Staubli VAL3: ros_server.pjx

--- ros_server.pjx ---
Parameters version=s8.12Cs9_BS2378 stackSize=5000 millimeterUnit=true
Program file=dataReceiver.pgx
Program file=dataStreamer.pgx
Program file=decodeMsgBody.pgx
Program file=decodeMsgHeader.pgx
Program file=decTrajPt.pgx
Program file=decTrajPtFull.pgx
Program file=encodeAck.pgx
Program file=encodeJState.pgx
Program file=encodeStatus.pgx
Program file=encPrefixHeader.pgx
Program file=encTrajPtAck.pgx
Program file=encTrajPtFAck.pgx
Program file=fetchStatus.pgx
Program file=initParams.pgx
Program file=interpolateVel.pgx
Program file=motionControl.pgx
Program file=pushMotion.pgx
Program file=recvData.pgx
Program file=recvHeartbeat.pgx
Program file=recvMsgBody.pgx
Program file=recvMsgHeader.pgx
Program file=recvTrajPt.pgx
Program file=recvTrajPtFull.pgx
Program file=screenUpdate.pgx
Program file=sendAck.pgx
Program file=sendData.pgx
Program file=sendRosMsg.pgx
Program file=setupRosMsgs.pgx
Program file=start.pgx
Program file=stop.pgx
Program file=taskManager.pgx
Program file=toJointArrayRad.pgx
Program file=toJointRxDeg.pgx
Data file=ros_server.dtx
Library alias=libQueueFuncs path=Disk://ros_libs/QueueFuncs/QueueFuncs.pjx
Library alias=libInterface path=Disk://ros_libs/UserInterface/interfaceDefault/interfaceDefault.pjx autoload=false
Type name=RosSimpleMsg path=Disk://ros_libs/RosSimpleMsg/RosSimpleMsg.pjx
Type name=RobotStatusMsg path=Disk://ros_libs/RobotStatusMsg/RobotStatusMsg.pjx
Type name=JointStateMsg path=Disk://ros_libs/JointStateMsg/JointStateMsg.pjx
Type name=JointTrajPtMsg path=Disk://ros_libs/JointTrajPtMsg/JointTrajPtMsg.pjx
Type name=JointTrajPtFMsg path=Disk://ros_libs/JointTrajPtFMsg/JointTrajPtFMsg.pjx
Type name=JointFbkMsg path=Disk://ros_libs/JointFbkMsg/JointFbkMsg.pjx
Type name=MotionCmd path=Disk://ros_libs/MotionCmd/MotionCmd.pjx
Type name=Header path=Disk://ros_libs/Header/Header.pjx
Type name=Prefix path=Disk://ros_libs/Prefix/Prefix.pjx
Type name=Body path=Disk://ros_libs/Body/Body.pjx
Type name=Queue path=Disk://ros_libs/Queue/Queue.pjx

--- ros_server.dtx ---
public bool bFbkOverrun
public bool bMotionOverrun
public sio siTcpIpFbk = {link=Socket\Feedback}
public sio siTcpIpMotion = {link=Socket\Motion}
public string sStreamTaskName = "publisher"
public string sMotionTaskName
public RosSimpleMsg rosGenericMsg
  [0]
    Header header
      [0]
        num nMsgType
        num nCommType
        num nReplyCode
        num nData[12]
    Prefix prefix
      [0]
        num nLength
        num nData[4]
public tool tTool = {fatherId=flange[0], ioLink=ValveIO\valve1}
public string sTrajPtTaskName
public bool bTrajPtOverrun
public RobotStatusMsg rosStatusMsg
  [0]
    Body body
      [0]
        num nData[28]
    Header header
      [0]
        num nMsgType
        num nCommType
        num nReplyCode
        num nData[12]
    Prefix prefix
      [0]
        num nLength
        num nData[4]
    RobotStatus robotStatus
      [0]
        num nDrivesPowered
        num nEStopped
        num nErrorCode
        num nInError
        num nInMotion
        num nMode
        num nMotionPossible
public JointStateMsg rosJointMsg
  [0]
    Header header
      [0]
        num nMsgType
        num nCommType
        num nReplyCode
        num nData[12]
    Body body
      [0]
        num nData[44]
    JointState jointState
      [0]
        num nSeq
        num nJoints[10]
    Prefix prefix
      [0]
        num nLength
        num nData[4]
public JointTrajPtMsg rosTrajPtMsg
  [0]
    Header header
      [0]
        num nMsgType
        num nCommType
        num nReplyCode
        num nData[12]
    JointTrajPt jointTrajPt
      [0]
        num nSeq
        num nJoints[10]
        num nVelocity
        num nDuration
    Prefix prefix
      [0]
        num nLength
        num nData[4]
    Body body
      [0]
        num nData[52]
public JointTrajPtFMsg rosTrajPtFMsg
  [0]
    Header header
      [0]
        num nMsgType
        num nCommType
        num nReplyCode
        num nData[12]
    Prefix prefix
      [0]
        num nLength
        num nData[4]
    JointTrajPtFull jointTrajPtFull
      [0]
        num nRobotId
        num nSeq
        num nValidFields
        num nTime
        num nPositions[10]
        num nVelocities[10]
        num nAccelerations[10]
    Body body
      [0]
        num nData[136]
public JointFbkMsg rosJointFbkMsg
  [0]
    Header header
      [0]
        num nMsgType
        num nCommType
        num nReplyCode
        num nData[12]
    Prefix prefix
      [0]
        num nLength
        num nData[4]
    JointFeedback jointFeedback
      [0]
        num nRobotId
        num nValidFields
        num nTime
        num nPositions[10]
        num nVelocities[10]
        num nAccelerations[10]
    Body body
      [0]
        num nData[132]
public JointTrajPtFMsg rosTrajPtFAck
  [0]
    Header header
      [0]
        num nMsgType
        num nCommType
        num nReplyCode
        num nData[12]
    Prefix prefix
      [0]
        num nLength
        num nData[4]
    JointTrajPtFull jointTrajPtFull
      [0]
        num nRobotId
        num nSeq
        num nValidFields
        num nTime
        num nPositions[10]
        num nVelocities[10]
        num nAccelerations[10]
    Body body
      [0]
        num nData[136]
public JointTrajPtMsg rosTrajPtAck
  [0]
    Header header
      [0]
        num nMsgType
        num nCommType
        num nReplyCode
        num nData[12]
    JointTrajPt jointTrajPt
      [0]
        num nSeq
        num nJoints[10]
        num nVelocity
        num nDuration
    Prefix prefix
      [0]
        num nLength
        num nData[4]
    Body body
      [0]
        num nData[52]
public bool bScreenOverrun
public string sScreenTaskName
public num nInConnFlag
public num nOutConnFlag
public string sHtbtTaskName
public num nPtsPopped
public bool bStopNow
public num nMotionProgress
public num nMoveId
public num nMovePts
public num nElapsedTime
public num nHeaderTime
public bool bOverwriteVel
public Queue qMoveBuffer
  [0]
    num nPush
    num nPop
    num nElems
    MotionCmd buffer[10]
      [0]
        mdesc mDesc = {leave=0, reach=0}
        num nDuration
        num nSequence
        jointRx jJointRx
      [1]
        mdesc mDesc = {leave=0, reach=0}
        num nDuration
        num nSequence
        jointRx jJointRx
      [2]
        mdesc mDesc = {leave=0, reach=0}
        num nDuration
        num nSequence
        jointRx jJointRx
      [3]
        mdesc mDesc = {leave=0, reach=0}
        num nDuration
        num nSequence
        jointRx jJointRx
      [4]
        mdesc mDesc = {leave=0, reach=0}
        num nDuration
        num nSequence
        jointRx jJointRx
      [5]
        mdesc mDesc = {leave=0, reach=0}
        num nDuration
        num nSequence
        jointRx jJointRx
      [6]
        mdesc mDesc = {leave=0, reach=0}
        num nDuration
        num nSequence
        jointRx jJointRx
      [7]
        mdesc mDesc = {leave=0, reach=0}
        num nDuration
        num nSequence
        jointRx jJointRx
      [8]
        mdesc mDesc = {leave=0, reach=0}
        num nDuration
        num nSequence
        jointRx jJointRx
      [9]
        mdesc mDesc = {leave=0, reach=0}
        num nDuration
        num nSequence
        jointRx jJointRx
public Queue qTrajPtBuffer
  [0]
    num nPush
    num nPop
    num nElems
    MotionCmd buffer[10]
      [0]
        mdesc mDesc = {leave=0, reach=0}
        num nDuration
        num nSequence
        jointRx jJointRx
      [1]
        mdesc mDesc = {leave=0, reach=0}
        num nDuration
        num nSequence
        jointRx jJointRx
      [2]
        mdesc mDesc = {leave=0, reach=0}
        num nDuration
        num nSequence
        jointRx jJointRx
      [3]
        mdesc mDesc = {leave=0, reach=0}
        num nDuration
        num nSequence
        jointRx jJointRx
      [4]
        mdesc mDesc = {leave=0, reach=0}
        num nDuration
        num nSequence
        jointRx jJointRx
      [5]
        mdesc mDesc = {leave=0, reach=0}
        num nDuration
        num nSequence
        jointRx jJointRx
      [6]
        mdesc mDesc = {leave=0, reach=0}
        num nDuration
        num nSequence
        jointRx jJointRx
      [7]
        mdesc mDesc = {leave=0, reach=0}
        num nDuration
        num nSequence
        jointRx jJointRx
      [8]
        mdesc mDesc = {leave=0, reach=0}
        num nDuration
        num nSequence
        jointRx jJointRx
      [9]
        mdesc mDesc = {leave=0, reach=0}
        num nDuration
        num nSequence
        jointRx jJointRx
num nVel[2]
num nStdMsgType{}
  [JOINT_TRAJ_PT] = 11
  [JOINT_TRAJ_PT_FULL] = 14
num nCommType{}
  [SERVICE_REQUEST] = 2
mdesc mNomSpeed
num nRecHeader
num nDecHeader = 1
num nRecBody = 2
num nDecBody = 3
num nPushMotion = 4
num nAck = 5
num nReset
num nFbkPeriod
num nMotionPeriod
num nTrajPeriod
num nScreenUpdate
num nFbkOverun
num nTrajPtOverrun
num nMotionOverrun
num nLibLoadError

--- start.pgx ---
program start()
  local num l_nScreenUpdate
  local string l_sVersionMajor
  local num l_nVersionMajor
  local bool l_bOkMajor
  local string l_sVersionMinor
  local num l_nVersionMinor
  local bool l_bOkMinor
  local num l_nLibLoad
begin
  // Copyright (c) 2016, Ocado Technology - Robotics Research Team
  //
  // Licensed under the Apache License, Version 2.0 (the "License");
  // you may not use this file except in compliance with the License.
  // You may obtain a copy of the License at
  //
  //     http://www.apache.org/licenses/LICENSE-2.0
  //
  // Unless required by applicable law or agreed to in writing, software
  // distributed under the License is distributed on an "AS IS" BASIS,
  // WITHOUT WARRANTIES OR CONDITIONS OF ANY KIND, either express or implied.
  // See the License for the specific language governing permissions and
  // limitations under the License.


  // Load interface library for CS8 or CS9
  //
  // CS9 handles the UI differently than CS8, requires
  // the UI funtions to be loaded in seperate libraries

  if(mid(getVersion("System"),1,1) == "7")
    // CS8 - VAL 3 rev 7
    // Check for VAL 3 version >= 7.7
    l_sVersionMajor = mid(getVersion("VAL3"),1,1)
    l_sVersionMinor = mid(getVersion("VAL3"),2,1)
    toNum(l_sVersionMajor, l_nVersionMajor, l_bOkMajor)
    toNum(l_sVersionMinor, l_nVersionMinor, l_bOkMinor)
    if(!l_bOkMajor or !l_bOkMinor)
      popUpMsg("Error reading VAL 3 version")
      call stop()
    endIf
    if( !((l_nVersionMajor == 7) and (l_nVersionMinor >= 7)))
      // VAL 3 version is too old
      popUpMsg("Error: VAL 3 version is < 7.7, socket communication will not work!")
      call stop()
    endIf
    nLibLoadError = libInterface:libLoad("ros_libs/UserInterface/interfaceCS8")
  elseIf(mid(getVersion("System"),1,1) == "8")
    // CS9 - VAL 3 rev 8
    nLibLoadError = libInterface:libLoad("ros_libs/UserInterface/interfaceCS9")
  endIf

  // check for libLoad error
  if nLibLoadError != 0
    popUpMsg("Error loading UserPage!")
    call stop()
  else
    // feedback task will run every 20ms (50Hz)
    nFbkPeriod=0.02
    //l_nFbkPeriod = 0.032 // 30Hz
    //l_nFbkPeriod = 0.05  // 20Hz
    //l_nFbkPeriod = 1.0   //  1Hz

    // motion control task will run every 4ms (250Hz)
    nMotionPeriod = 0.004
    //l_nMotionPeriod=0.012  // 83Hz
    //l_nMotionPeriod = 0.05 // 20Hz

    // data (trajectory) reception task will run every 4ms (250Hz)
    nTrajPeriod = 0.004
    // not in use at the moment
    nScreenUpdate = 1.0

    sStreamTaskName = "streamerTask"
    sTrajPtTaskName = "trajPtTask"
    sMotionTaskName = "motionTask"
    sScreenTaskName = "screenTask"
    sHtbtTaskName = "htbtTask"

    // initialise TCP/IP parameters
    call initParams()
    // setup prefix and header of ROS messages
    call setupRosMsgs()

    // socket connection status flags: initially disconnected
    nInConnFlag = 0
    nOutConnFlag = 0

    // flag defining whether velocity to be overwritten to max. vel.
    bOverwriteVel = false

    nPtsPopped = 0
    nMovePts = 0

    // flush buffer of incoming socket
    clearBuffer(siTcpIpMotion)
    // flush buffer of outgoing socket
    clearBuffer(siTcpIpFbk)

    // check if robot is not in emergency stop and wait until estop is reset
    if(esStatus() == 2)
      popUpMsg("Please reset E-Stop")
      wait(esStatus() < 2)
    endIf

    // before anything else, enable power (only works if robot is in remote mode)
    if(!isPowered())
      if(workingMode() >= 4)
        do
          enablePower()
          delay(2)
        until isPowered()
      else
        popUpMsg("Power must be enabled manually")
      endIf
    endIf

    // reset motion, potentially setting a start joint position for calling autoConnect() in the future
    resetMotion()

    //start task for the taskManager:
    taskCreate "taskManager", 50, taskManager()
    wait(taskStatus("taskManager") != -1)
  endIf


end

--- dataReceiver.pgx ---
public program dataReceiver()
  local num l_nStartTime
  local num l_nMsgRecvState
begin
  // Copyright (c) 2016, Ocado Technology - Robotics Research Team
  //
  // Licensed under the Apache License, Version 2.0 (the "License");
  // you may not use this file except in compliance with the License.
  // You may obtain a copy of the License at
  //
  //     http://www.apache.org/licenses/LICENSE-2.0
  //
  // Unless required by applicable law or agreed to in writing, software
  // distributed under the License is distributed on an "AS IS" BASIS,
  // WITHOUT WARRANTIES OR CONDITIONS OF ANY KIND, either express or implied.
  // See the License for the specific language governing permissions and
  // limitations under the License.



  // state machine at initial state
  // 0: receive header
  // 1: decode header
  // 2: receive body
  // 3: decode body
  // 4: push motion into buffer
  // 5: send ACK

  // Set variable constants to make sure they were not changed
  nReset=0
  nRecHeader=0
  nDecHeader=1
  nRecBody=2
  nDecBody=3
  nPushMotion=4
  nAck=5

  l_nMsgRecvState=nRecHeader

  while(true)
    // usually for state machines a switch-case statement is a neat implementation
    // HOWEVER, at every iteration of while() this task is sequenced and only called
    // after whatever ms is was defined when created.
    // As a result, receiving one single message, pushing motion and sending ACK
    // would take 6 * task period using switch-case statement.
    // The desirable behaviour is to receive and decode a full message, push motion
    // into buffer and then send ACK to client WITHIN ONE ITERATION of while(),
    // hence the if statement sequence below

        // check for overrun
    if bTrajPtOverrun
      nTrajPtOverrun = nTrajPtOverrun + 1
    endIf


    l_nStartTime = clock()
    if(l_nMsgRecvState==nRecHeader)
      call recvMsgHeader(l_nMsgRecvState)
    endIf
    nHeaderTime = clock() - l_nStartTime
    if(l_nMsgRecvState==nDecHeader)
      call decodeMsgHeader(l_nMsgRecvState)
    endIf
    if(l_nMsgRecvState==nRecBody)
      call recvMsgBody(l_nMsgRecvState)
    endIf
    if(l_nMsgRecvState==nDecBody)
      call decodeMsgBody(l_nMsgRecvState)
    endIf
    if(l_nMsgRecvState==nPushMotion)
      call pushMotion(l_nMsgRecvState)
    endIf
    if(l_nMsgRecvState==nAck)
      call encodeAck()
      call sendAck(l_nMsgRecvState)
    endIf
    nElapsedTime = clock() - l_nStartTime - nHeaderTime

    // assert state machine is working OK
    if(l_nMsgRecvState<nRecHeader or l_nMsgRecvState>nAck)
      popUpMsg("Data reception state machine error")
    endIf

    // sequence task
    delay(0)


  endWhile
end

--- dataStreamer.pgx ---
public program dataStreamer()
  local num l_nThrottle
  local jointRx l_jCurrPose
begin
  // Copyright (c) 2016, Ocado Technology - Robotics Research Team
  //
  // Licensed under the Apache License, Version 2.0 (the "License");
  // you may not use this file except in compliance with the License.
  // You may obtain a copy of the License at
  //
  //     http://www.apache.org/licenses/LICENSE-2.0
  //
  // Unless required by applicable law or agreed to in writing, software
  // distributed under the License is distributed on an "AS IS" BASIS,
  // WITHOUT WARRANTIES OR CONDITIONS OF ANY KIND, either express or implied.
  // See the License for the specific language governing permissions and
  // limitations under the License.



  l_nThrottle = 0
  while(true)
    // check for overrun
    if bFbkOverrun
      nFbkOverun = nFbkOverun + 1
    endIf

    // only attempt to send data if flag indicates that connection is established
      if(nOutConnFlag == 1)
        // fetch current joint positions
        l_jCurrPose=herej()
        // encode and send ROS simple_message ID 10: joint state
        call encodeJState(l_jCurrPose)
        call sendRosMsg(siTcpIpFbk, rosJointMsg.prefix, rosJointMsg.header, rosJointMsg.body, nOutConnFlag)

        // send Robot Status messages 5 times slower than Joint State
        if(l_nThrottle == 5)
          // fetch robot status
          call fetchStatus()
          // encode and send ROS simple_message ID 13: robot status
          call encodeStatus()
          call sendRosMsg(siTcpIpFbk, rosStatusMsg.prefix, rosStatusMsg.header, rosStatusMsg.body, nOutConnFlag)
          l_nThrottle = 0
        endIf
        l_nThrottle = l_nThrottle + 1
      else
        delay(0.1)
      endIf

      // sequence task
      delay(0)
  endWhile
end

--- decodeMsgBody.pgx ---
public program decodeMsgBody(RosSimpleMsg& x_msg, num& x_nMsgRecvState)
  local bool l_bFlag
begin
  // Copyright (c) 2016, Ocado Technology - Robotics Research Team
  // Copyright (c) 2021, Institute for Factory Automation and Production Systems (FAPS)
  //
  // Licensed under the Apache License, Version 2.0 (the "License");
  // you may not use this file except in compliance with the License.
  // You may obtain a copy of the License at
  //
  //     http://www.apache.org/licenses/LICENSE-2.0
  //
  // Unless required by applicable law or agreed to in writing, software
  // distributed under the License is distributed on an "AS IS" BASIS,
  // WITHOUT WARRANTIES OR CONDITIONS OF ANY KIND, either express or implied.
  // See the License for the specific language governing permissions and
  // limitations under the License.


  // assume failure to decode
  l_bFlag=false

  //region @decode -- call specific decode function
  switch x_msg.header.nMsgType
    case SimpleMsg:MsgType.JOINT_TRAJ_PT
      call decTrajPt(l_bFlag)
    break
    case SimpleMsg:MsgType.JOINT_TRAJ_PT_F
      call decTrajPtFull(l_bFlag)
    break
    // Staubli specific
    case Staubli:MsgType.SET_DRIVE_POWER
      call Staubli:decSetDrvPwrMsg(l_bFlag)
    break
    case Staubli:MsgType.WRITE_SINGLE_IO
      call Staubli:decWriSingIOMsg(l_bFlag)
    break
    case Staubli:MsgType.VELOCITY_CFG
      call Staubli:decodeVelCfg(l_bFlag)
    break
    case Staubli:MsgType.VELOCITY_CMD
      call Staubli:decodeVelCmd(l_bFlag)
    break
    default
      //region @DEBUG
      if (bDebugMode and nDebugLevel<=3)
        call printDebug("ERROR: unknown msg type ("+toString("",x_msg.header.nMsgType)+")",false)
        call printDebug("       could not decode message",false)
      endIf
      //endregion
    break
  endSwitch
  //endregion

  //region @check_success -- check whether decoding was successful and move on to the next state
  if (l_bFlag == true)
    switch x_msg.header.nMsgType
      case SimpleMsg:MsgType.JOINT_TRAJ_PT,SimpleMsg:MsgType.JOINT_TRAJ_PT_F,Staubli:MsgType.VELOCITY_CFG,Staubli:MsgType.VELOCITY_CMD
        // move on to state: push motion into buffer
        x_nMsgRecvState = MsgRecvState.PUSH_MOTION
      break
      case Staubli:MsgType.SET_DRIVE_POWER, Staubli:MsgType.WRITE_SINGLE_IO
        // move on to state: handle system/io request
        x_nMsgRecvState = MsgRecvState.HANDLE_REQUEST
      break
    endSwitch

    //region @DEBUG
    if (bDebugMode and nDebugLevel<=3)
      call printDebug("INFO: decoding successful",false)
    endIf
    //endregion
  else
    // error whilst decoding msg body...
    if (x_msg.header.nCommType==SimpleMsg:CommType.SERVICE_REQUEST)
      // set reply code if comm type is request
      switch x_msg.header.nMsgType
        case SimpleMsg:MsgType.JOINT_TRAJ_PT
          rosTrajPtAck.header.nReplyCode=SimpleMsg:ReplyCode.FAILURE
        break
        case SimpleMsg:MsgType.JOINT_TRAJ_PT_F
          rosTrajPtFAck.header.nReplyCode=SimpleMsg:ReplyCode.FAILURE
        break
        // Staubli specific
        case Staubli:MsgType.SET_DRIVE_POWER
          Staubli:setDrvPwrAck.header.nReplyCode=SimpleMsg:ReplyCode.FAILURE
        break
        case Staubli:MsgType.WRITE_SINGLE_IO
          Staubli:writeSingIOAck.header.nReplyCode=SimpleMsg:ReplyCode.FAILURE
        break
        case Staubli:MsgType.VELOCITY_CFG
          Staubli:velCfgAck.header.nReplyCode=SimpleMsg:ReplyCode.FAILURE
        break
        case Staubli:MsgType.VELOCITY_CMD
          Staubli:velCmdAck.header.nReplyCode=SimpleMsg:ReplyCode.FAILURE
        break
        default
          //region @DEBUG
          if (bDebugMode and nDebugLevel<=3)
            call printDebug("ERROR: unknown msg type ("+toString("",x_msg.header.nMsgType)+")",false)
            call printDebug("       could not set reply code",false)
          endIf
          //endregion
        break
      endSwitch
      // jump to state 6: sendAck()
      x_nMsgRecvState = MsgRecvState.SEND_ACK
    else
      // reset state machine, since no ACK is required
      x_nMsgRecvState = MsgRecvState.RECEIVE_HEADER
    endIf
    //region @DEBUG
    if (bDebugMode and nDebugLevel<=3)
      call printDebug("ERROR: decoding not successful",false)
    endIf
    //endregion
  endIf
  //endregion
end

--- decodeMsgHeader.pgx ---
public program decodeMsgHeader(RosSimpleMsg& x_msg (dimensions=1), num& x_nMsgRecvState (dimensions=1))
  local num l_nRetVal
begin
  // Copyright (c) 2016, Ocado Technology - Robotics Research Team
  // Copyright (c) 2021, Institute for Factory Automation and Production Systems (FAPS)
  //
  // Licensed under the Apache License, Version 2.0 (the "License");
  // you may not use this file except in compliance with the License.
  // You may obtain a copy of the License at
  //
  //     http://www.apache.org/licenses/LICENSE-2.0
  //
  // Unless required by applicable law or agreed to in writing, software
  // distributed under the License is distributed on an "AS IS" BASIS,
  // WITHOUT WARRANTIES OR CONDITIONS OF ANY KIND, either express or implied.
  // See the License for the specific language governing permissions and
  // limitations under the License.



  // decode message into generic message first
  l_nRetVal=fromBinary(x_msg.prefix.nData,4,"-4l",x_msg.prefix.nLength)
  if (l_nRetVal!=1)
    // error decoding prefix, reset state machine
    x_nMsgRecvState = MsgRecvState.RECEIVE_HEADER
    return
  endIf
  l_nRetVal=fromBinary(x_msg.header.nData,4,"-4l",x_msg.header.nMsgType)
  if (l_nRetVal!=1)
    // error decoding header (msg type), reset state machine
    x_nMsgRecvState = MsgRecvState.RECEIVE_HEADER
    return
  endIf
  l_nRetVal=fromBinary(x_msg.header.nData[4],4,"-4l",x_msg.header.nCommType)
  if (l_nRetVal!=1)
    // error decoding header (comm type), reset state machine
    x_nMsgRecvState = MsgRecvState.RECEIVE_HEADER
    return
  endIf
  l_nRetVal=fromBinary(x_msg.header.nData[8],4,"-4l",x_msg.header.nReplyCode)
  if (l_nRetVal!=1)
    // error decoding header (reply code), reset state machine
    x_nMsgRecvState = MsgRecvState.RECEIVE_HEADER
    return
  endIf

  // no errors detected whilst decoding prefix and header
  // move on to state 2: receive msg body
  x_nMsgRecvState = MsgRecvState.RECEIVE_BODY

  // debug
  if (bDebugMode and nDebugLevel<=1)
    call printDebug("decodeMsgHeader: successful",true)
    call printDebug("Prefix    :"+toString("",x_msg.prefix.nLength),false)
    call printDebug("MsgType   :"+toString("",x_msg.header.nMsgType),false)
    call printDebug("CommType  :"+toString("",x_msg.header.nCommType),false)
    call printDebug("ReplyType :"+toString("",x_msg.header.nReplyCode),false)
  endIf
end

--- decTrajPt.pgx ---
public program decTrajPt(bool& x_bFlag)
  local num l_nIndex
  local num l_nRetVal
begin
  // Copyright (c) 2016, Ocado Technology - Robotics Research Team
  //
  // Licensed under the Apache License, Version 2.0 (the "License");
  // you may not use this file except in compliance with the License.
  // You may obtain a copy of the License at
  //
  //     http://www.apache.org/licenses/LICENSE-2.0
  //
  // Unless required by applicable law or agreed to in writing, software
  // distributed under the License is distributed on an "AS IS" BASIS,
  // WITHOUT WARRANTIES OR CONDITIONS OF ANY KIND, either express or implied.
  // See the License for the specific language governing permissions and
  // limitations under the License.



  // decode message ID 11 body (data)

  // assume failure to decode
  rosTrajPtAck.header.nReplyCode=2

  // sequence
  l_nRetVal=fromBinary(rosTrajPtMsg.body.nData,4,"-4l",rosTrajPtMsg.jointTrajPt.nSeq)
  if(l_nRetVal!=1)
    x_bFlag=false
    return
  endIf

  // joints[10]
  for l_nIndex=0 to 9 step 1
    l_nRetVal=fromBinary(rosTrajPtMsg.body.nData[(l_nIndex*4)+4],4,"4.0l",rosTrajPtMsg.jointTrajPt.nJoints[l_nIndex])
    if(l_nRetVal!=1)
      x_bFlag=false
      return
    endIf
  endFor

  // velocity
  l_nRetVal=fromBinary(rosTrajPtMsg.body.nData[44],4,"4.0l",rosTrajPtMsg.jointTrajPt.nVelocity)
  if(l_nRetVal!=1)
    x_bFlag=false
    return
  endIf

  // duration
  l_nRetVal=fromBinary(rosTrajPtMsg.body.nData[48],4,"4.0l",rosTrajPtMsg.jointTrajPt.nDuration)
  if(l_nRetVal!=1)
    x_bFlag=false
    return
  endIf

  // decoding successful
  rosTrajPtAck.header.nReplyCode=1
  rosTrajPtAck.jointTrajPt.nSeq=rosTrajPtMsg.jointTrajPt.nSeq
  x_bFlag=true
end

--- decTrajPtFull.pgx ---
public program decTrajPtFull(bool& x_bFlag)
  local num l_nIndex
  local num l_nRetVal
begin
  // Copyright (c) 2016, Ocado Technology - Robotics Research Team
  //
  // Licensed under the Apache License, Version 2.0 (the "License");
  // you may not use this file except in compliance with the License.
  // You may obtain a copy of the License at
  //
  //     http://www.apache.org/licenses/LICENSE-2.0
  //
  // Unless required by applicable law or agreed to in writing, software
  // distributed under the License is distributed on an "AS IS" BASIS,
  // WITHOUT WARRANTIES OR CONDITIONS OF ANY KIND, either express or implied.
  // See the License for the specific language governing permissions and
  // limitations under the License.



  // decode message ID 14 body (data)

  // assume failure to decode
  rosTrajPtFAck.header.nReplyCode=2

  // robotId
  l_nRetVal=fromBinary(rosTrajPtFMsg.body.nData,4,"-4l",rosTrajPtFMsg.jointTrajPtFull.nRobotId)
  if(l_nRetVal!=1)
    x_bFlag=false
    return
  endIf

  // sequence
  l_nRetVal=fromBinary(rosTrajPtFMsg.body.nData,4,"-4l",rosTrajPtFMsg.jointTrajPtFull.nSeq)
  if(l_nRetVal!=1)
    x_bFlag=false
    return
  endIf

  // valid fields
  l_nRetVal=fromBinary(rosTrajPtFMsg.body.nData,4,"-4l",rosTrajPtFMsg.jointTrajPtFull.nValidFields)
  if(l_nRetVal!=1)
    x_bFlag=false
    return
  endIf

  // time
  l_nRetVal=fromBinary(rosTrajPtFMsg.body.nData,4,"4.0l",rosTrajPtFMsg.jointTrajPtFull.nTime)
  if(l_nRetVal!=1)
    x_bFlag=false
    return
  endIf

  // positions[10]
  for l_nIndex=0 to 9 step 1
    l_nRetVal=fromBinary(rosTrajPtFMsg.body.nData[(l_nIndex*4)+16],4,"4.0l",rosTrajPtFMsg.jointTrajPtFull.nPositions[l_nIndex])
    if(l_nRetVal!=1)
      x_bFlag=false
      return
    endIf
  endFor

  // velocities[10]
  for l_nIndex=0 to 9 step 1
    l_nRetVal=fromBinary(rosTrajPtFMsg.body.nData[(l_nIndex*4)+56],4,"4.0l",rosTrajPtFMsg.jointTrajPtFull.nVelocities[l_nIndex])
    if(l_nRetVal!=1)
      x_bFlag=false
      return
    endIf
  endFor

  // accelerations[10]
  for l_nIndex=0 to 9 step 1
    l_nRetVal=fromBinary(rosTrajPtFMsg.body.nData[(l_nIndex*4)+96],4,"4.0l",rosTrajPtFMsg.jointTrajPtFull.nAccelerations[l_nIndex])
    if(l_nRetVal!=1)
      x_bFlag=false
      return
    endIf
  endFor

  // decoding successful
  rosTrajPtFAck.header.nReplyCode=1
  rosTrajPtFAck.jointTrajPtFull.nSeq=rosTrajPtFMsg.jointTrajPtFull.nSeq
  x_bFlag=true
end

--- encodeAck.pgx ---
public program encodeAck(RosSimpleMsg& x_msg)
begin
  // Copyright (c) 2016, Ocado Technology - Robotics Research Team
  // Copyright (c) 2021, Institute for Factory Automation and Production Systems (FAPS)
  //
  // Licensed under the Apache License, Version 2.0 (the "License");
  // you may not use this file except in compliance with the License.
  // You may obtain a copy of the License at
  //
  //     http://www.apache.org/licenses/LICENSE-2.0
  //
  // Unless required by applicable law or agreed to in writing, software
  // distributed under the License is distributed on an "AS IS" BASIS,
  // WITHOUT WARRANTIES OR CONDITIONS OF ANY KIND, either express or implied.
  // See the License for the specific language governing permissions and
  // limitations under the License.



  switch x_msg.header.nMsgType

    case SimpleMsg:MsgType.JOINT_TRAJ_PT
      call encTrajPtAck()
    break

    case SimpleMsg:MsgType.JOINT_TRAJ_PT_F
      call encTrajPtFAck()
    break

    // Staubli specific
    case Staubli:MsgType.SET_DRIVE_POWER
      call Staubli:encSetDrvPwrAck()
    break

    case Staubli:MsgType.WRITE_SINGLE_IO
      call Staubli:encWriSingIOAck()
    break

    case Staubli:MsgType.VELOCITY_CFG
      call Staubli:encodeVelCfgAck()
    break

    case Staubli:MsgType.VELOCITY_CMD
      call Staubli:encodeVelCmdAck()
    break

    default
      //region @DEBUG
      if (bDebugMode and nDebugLevel<=5)
        call printDebug("encodeAck: switch (msgType)",true)
        call printDebug("ERROR: unknown msg type",false)
      endIf
      //endregion
    break
  endSwitch
end

--- encodeJFeedback.pgx ---
program encodeJFeedback(num x_nTime, jointRx x_jPosition, jointRx x_jVelocity)
begin
  // Copyright (c) 2021, Institute for Factory Automation and Production Systems (FAPS)
  //
  // Licensed under the Apache License, Version 2.0 (the "License");
  // you may not use this file except in compliance with the License.
  // You may obtain a copy of the License at
  //
  //     http://www.apache.org/licenses/LICENSE-2.0
  //
  // Unless required by applicable law or agreed to in writing, software
  // distributed under the License is distributed on an "AS IS" BASIS,
  // WITHOUT WARRANTIES OR CONDITIONS OF ANY KIND, either express or implied.
  // See the License for the specific language governing permissions and
  // limitations under the License.


  // encode 'prefix' and 'header'
  call encPrefixHeader(rosJointFbkMsg.prefix, rosJointFbkMsg.header)

  // encode 'robot_id' variable of body message (data)
  toBinary(rosJointFbkMsg.jointFeedback.nRobotId, 1, "-4l", rosJointFbkMsg.body.nData)

  // encode 'valid_fields' variable of body message (data)
  toBinary(rosJointFbkMsg.jointFeedback.nValidFields, 1, "-4l", rosJointFbkMsg.body.nData[4])

  // encode 'time' variable of body message (data)
  toBinary(rosJointFbkMsg.jointFeedback.nTime, 1, "-4l", rosJointFbkMsg.body.nData[8])

  call toJointArrayRad(x_jPosition, rosJointFbkMsg.jointFeedback.nPositions)

  // encode 10 values representing joint positions [10]
  toBinary(rosJointFbkMsg.jointFeedback.nPositions, 10, "4.0l", rosJointFbkMsg.body.nData[12])

  call toJointArrayRad(x_jVelocity, rosJointFbkMsg.jointFeedback.nVelocities)

  // encode 10 values representing joint velocities [10]
  toBinary(rosJointFbkMsg.jointFeedback.nVelocities, 10, "4.0l", rosJointFbkMsg.body.nData[52])
end

--- fetchStatus.pgx ---
public program fetchStatus()
begin
  // Copyright (c) 2016, Ocado Technology - Robotics Research Team
  // Copyright (c) 2021, Institute for Factory Automation and Production Systems (FAPS)
  //
  // Licensed under the Apache License, Version 2.0 (the "License");
  // you may not use this file except in compliance with the License.
  // You may obtain a copy of the License at
  //
  //     http://www.apache.org/licenses/LICENSE-2.0
  //
  // Unless required by applicable law or agreed to in writing, software
  // distributed under the License is distributed on an "AS IS" BASIS,
  // WITHOUT WARRANTIES OR CONDITIONS OF ANY KIND, either express or implied.
  // See the License for the specific language governing permissions and
  // limitations under the License.



  // fetch robot status data

  // drives_powered
  if (isPowered()==true)
    rosStatusMsg.robotStatus.nDrivesPowered=1
  else
    rosStatusMsg.robotStatus.nDrivesPowered=0
  endIf

  // e-stopped
  if (esStatus()==2)
    rosStatusMsg.robotStatus.nEStopped=1
  else
    rosStatusMsg.robotStatus.nEStopped=0
  endIf

  // error_code
  if (taskStatus(sMotionTask) > 1)
    rosStatusMsg.robotStatus.nErrorCode = taskStatus(sMotionTask)
  elseIf (taskStatus(sMotionRecvTask) > 1)
    rosStatusMsg.robotStatus.nErrorCode = taskStatus(sMotionRecvTask)
  elseIf (taskStatus(sStreamerTask) > 1)
    rosStatusMsg.robotStatus.nErrorCode = taskStatus(sStreamerTask)
  elseIf (taskStatus(sHeartbeatTask) > 1)
    rosStatusMsg.robotStatus.nErrorCode = taskStatus(sHeartbeatTask)
  elseIf (taskStatus(sScreenTask) > 1)
    rosStatusMsg.robotStatus.nErrorCode = taskStatus(sScreenTask)
  else
    rosStatusMsg.robotStatus.nErrorCode = 0
  endIf

  // in_error
  if (taskStatus(sMotionRecvTask) == 1 and taskStatus(sMotionTask) == 1 and taskStatus(sStreamerTask) == 1 and taskStatus(sScreenTask) == 1 and taskStatus(sHeartbeatTask) == 1)
    rosStatusMsg.robotStatus.nInError = 0
  else
    rosStatusMsg.robotStatus.nInError = 1
  endIf

  // in_motion
  if (isSettled()==true)
    rosStatusMsg.robotStatus.nInMotion=0
  else
    rosStatusMsg.robotStatus.nInMotion=1
  endIf

  // mode (controller/pendant mode)
  // according to industrial_msgs/RobotMode, possible values are:
  // -1: unknown or unavailable
  //  1: teach or manual mode
  //  2: automatic mode (which I interpret as either local or remote)
  if (workingMode() == 0)
    rosStatusMsg.robotStatus.nMode = -1
  elseIf (workingMode()==1 or workingMode()==2)
    rosStatusMsg.robotStatus.nMode = 1
  elseIf (workingMode()==3 or workingMode()==4)
    rosStatusMsg.robotStatus.nMode = 2
  endIf

  // motion_possible:
  // drives must be powered and e-stop must be off
  // and dataReceiver and motionControl tasks must be
  // running normally
  if (isPowered() == true and esStatus() == 0 and taskStatus(sMotionRecvTask) == 1 and taskStatus(sMotionTask) == 1)
    rosStatusMsg.robotStatus.nMotionPossible=1
  else
    rosStatusMsg.robotStatus.nMotionPossible=0
  endIf
end

--- handleRequest.pgx ---
public program handleRequest(RosSimpleMsg& x_msg, num& x_nMsgRecvState)
  local bool l_bOk
  local num l_nModuleId
  local num l_nPin
  local bool l_bState
begin
  // Copyright (c) 2021, Institute for Factory Automation and Production Systems (FAPS)
  //
  // Licensed under the Apache License, Version 2.0 (the "License");
  // you may not use this file except in compliance with the License.
  // You may obtain a copy of the License at
  //
  //     http://www.apache.org/licenses/LICENSE-2.0
  //
  // Unless required by applicable law or agreed to in writing, software
  // distributed under the License is distributed on an "AS IS" BASIS,
  // WITHOUT WARRANTIES OR CONDITIONS OF ANY KIND, either express or implied.
  // See the License for the specific language governing permissions and
  // limitations under the License.


  // assume success to push motion
  l_bOk=true

  // handle request
  switch x_msg.header.nMsgType
    case Staubli:MsgType.SET_DRIVE_POWER
      if (Staubli:setDrvPwrMsg.bDrivePower==true and isPowered()==false)
        enablePower()
      elseIf (Staubli:setDrvPwrMsg.bDrivePower==false and isPowered()==true)
        disablePower()
      else
        // nothing to do
      endIf
    break
    case Staubli:MsgType.WRITE_SINGLE_IO
      l_nModuleId=Staubli:writeSingIOMsg.writeSingleIO.nModuleId
      l_nPin=Staubli:writeSingIOMsg.writeSingleIO.nPin
      l_bState=Staubli:writeSingIOMsg.writeSingleIO.bState
      call IO:writeSingle(l_nModuleId,l_nPin,l_bState,l_bOk)
    break
    // unknown message type
    default
      l_bOk=false
      //region @DEBUG
      if (bDebugMode and nDebugLevel<=4)
        call printDebug("ERROR: unknown msg type ("+toString("",x_msg.header.nMsgType)+")",false)
      endIf
      //endregion
    break
  endSwitch

  //region @check_success -- check whether handling request was successful
  if (l_bOk)
    //region @DEBUG
    if (bDebugMode and nDebugLevel<=4)
      call printDebug("INFO: handling request successful",false)
    endIf
    //endregion
  else
    // could not handle request
    // thus ACK should flag FAILURE, but only if comm type is request
    if (x_msg.header.nCommType==SimpleMsg:CommType.SERVICE_REQUEST)
      switch x_msg.header.nMsgType
        case Staubli:MsgType.SET_DRIVE_POWER
          Staubli:setDrvPwrAck.header.nReplyCode=SimpleMsg:ReplyCode.FAILURE
        break
        case Staubli:MsgType.WRITE_SINGLE_IO
          Staubli:writeSingIOAck.header.nReplyCode=SimpleMsg:ReplyCode.FAILURE
        break
        default
        break
      endSwitch
    endIf
    //region @DEBUG
    if (bDebugMode and nDebugLevel<=4)
      call printDebug("ERROR: handling request not successful",false)
    endIf
    //endregion
  endIf
  //endregion

  //region @check_reply -- check whether service reply (ACK) should be sent
  if (x_msg.header.nCommType==SimpleMsg:CommType.SERVICE_REQUEST)
    // comm type request requires ACK
    x_nMsgRecvState = MsgRecvState.SEND_ACK
  else
    // other comm types (e.g., topic) does not require ACK, hence skip state
    x_nMsgRecvState = MsgRecvState.RECEIVE_HEADER
  endIf
  //endregion
end

--- initParams.pgx ---
public program initParams()
  local num l_nRetVal
begin
  // Copyright (c) 2016, Ocado Technology - Robotics Research Team
  // Copyright (c) 2021, Institute for Factory Automation and Production Systems (FAPS)
  //
  // Licensed under the Apache License, Version 2.0 (the "License");
  // you may not use this file except in compliance with the License.
  // You may obtain a copy of the License at
  //
  //     http://www.apache.org/licenses/LICENSE-2.0
  //
  // Unless required by applicable law or agreed to in writing, software
  // distributed under the License is distributed on an "AS IS" BASIS,
  // WITHOUT WARRANTIES OR CONDITIONS OF ANY KIND, either express or implied.
  // See the License for the specific language governing permissions and
  // limitations under the License.

  MsgRecvState.RECEIVE_HEADER=0
  MsgRecvState.DECODE_HEADER=1
  MsgRecvState.RECEIVE_BODY=2
  MsgRecvState.DECODE_BODY=3
  MsgRecvState.PUSH_MOTION=4
  MsgRecvState.HANDLE_REQUEST=5
  MsgRecvState.SEND_ACK=6

  l_nRetVal=sioCtrl(siTcpIpIO,"timeout",-1)
  if (l_nRetVal!=0)
    popUpMsg("Error while setting 'IO' socket timeout")
  endIf

  l_nRetVal=sioCtrl(siTcpIpMotion,"timeout",-1)
  if (l_nRetVal!=0)
    popUpMsg("Error while setting 'Motion' socket timeout")
  endIf

  l_nRetVal=sioCtrl(siTcpIpState,"timeout",-1)
  if (l_nRetVal!=0)
    popUpMsg("Error while setting 'State' socket timeout")
  endIf

  l_nRetVal=sioCtrl(siTcpIpSystem,"timeout",-1)
  if (l_nRetVal!=0)
    popUpMsg("Error while setting 'System' socket timeout")
  endIf
end

--- initRosMsgs.pgx ---
public program initRosMsgs()
begin
  // Copyright (c) 2016, Ocado Technology - Robotics Research Team
  //
  // Licensed under the Apache License, Version 2.0 (the "License");
  // you may not use this file except in compliance with the License.
  // You may obtain a copy of the License at
  //
  //     http://www.apache.org/licenses/LICENSE-2.0
  //
  // Unless required by applicable law or agreed to in writing, software
  // distributed under the License is distributed on an "AS IS" BASIS,
  // WITHOUT WARRANTIES OR CONDITIONS OF ANY KIND, either express or implied.
  // See the License for the specific language governing permissions and
  // limitations under the License.



  // Joint state message (ID 10)
  // prefix length = 12 + 44
  rosJointMsg.prefix.nLength=56
  rosJointMsg.header.nMsgType=10
  rosJointMsg.header.nCommType=1
  rosJointMsg.header.nReplyCode=0
  // sequence
  rosJointMsg.jointState.nSeq=0



  // Trajectory point message (ID 11)
  // prefix length = 12 + 52
  rosTrajPtAck.prefix.nLength=64
  rosTrajPtAck.header.nMsgType=11
  rosTrajPtAck.header.nCommType=3
  // reply: 1 = success, 2 = failure
  rosTrajPtAck.header.nReplyCode=1
  // joints are assumed to be initiliased to zero

  // the message bellow will be filled upon reception
  rosTrajPtMsg.prefix.nLength=64



  // Robot status message (ID 13)
  // prefix length = 12 + 28
  rosStatusMsg.prefix.nLength=40
  rosStatusMsg.header.nMsgType=13
  rosStatusMsg.header.nCommType=1
  rosStatusMsg.header.nReplyCode=0



  // Trajectory point full message (ID 14)
  // prefix length = 12 + 136
  rosTrajPtFAck.prefix.nLength=148
  rosTrajPtFAck.header.nMsgType=14
  rosTrajPtFAck.header.nCommType=3
  // reply: 1 = success, 2 = failure
  rosTrajPtFAck.header.nReplyCode=1
  // body (data) assumed to be initialised to zero

  // the message bellow will be filled upon reception
  rosTrajPtFMsg.prefix.nLength=148



  // Joint feedback message (ID 15)
  // prefix length = 12 + 132
  rosJointFbkMsg.prefix.nLength=144
  rosJointFbkMsg.header.nMsgType=15
  rosJointFbkMsg.header.nCommType=1
  rosJointFbkMsg.header.nReplyCode=0
end

--- interpolateVel.pgx ---
program interpolateVel(MotionCmd x_mMotion)
begin
  // Applies velocity "smoothing" to last point in trajectory when vel==0 is replaced by vel==0.1 (default for MoveIt)

  // Round to remove trailing decimal places from fromBinary()
  x_mMotion.mDesc.vel = x_mMotion.mDesc.vel * 10000
  x_mMotion.mDesc.vel = round(x_mMotion.mDesc.vel)
  x_mMotion.mDesc.vel = x_mMotion.mDesc.vel / 10000
  // Smooth last point in traj
  if((x_mMotion.mDesc.vel == 0.1) and (x_mMotion.nSequence != 0))
    x_mMotion.mDesc.vel = (nVel[0] - (nVel[1] - nVel[0]))
  endIf

end

--- motionControl.pgx ---
public program motionControl()
  local MotionCmd l_mTrajPt
  local bool l_bFlag
  local MotionCmd l_motion
  local num l_nElems
begin
  // Copyright (c) 2016, Ocado Technology - Robotics Research Team
  //
  // Licensed under the Apache License, Version 2.0 (the "License");
  // you may not use this file except in compliance with the License.
  // You may obtain a copy of the License at
  //
  //     http://www.apache.org/licenses/LICENSE-2.0
  //
  // Unless required by applicable law or agreed to in writing, software
  // distributed under the License is distributed on an "AS IS" BASIS,
  // WITHOUT WARRANTIES OR CONDITIONS OF ANY KIND, either express or implied.
  // See the License for the specific language governing permissions and
  // limitations under the License.



  nMoveId = -1

  while(true)

    if bMotionOverrun
      nMotionOverrun = nMotionOverrun + 1
    endIf

    // check connection status, and whether to stop motion
    if(nInConnFlag == 1 and nOutConnFlag == 1 and bStopNow == false)

      // process trajectory point from trajectory buffer
      call libQueueFuncs:getNumElems(qTrajPtBuffer, l_nElems)
      if(l_nElems > 0)
        call libQueueFuncs:pop(qTrajPtBuffer,l_mTrajPt, l_bFlag)
        if(l_bFlag == true)
          nPtsPopped = nPtsPopped + 1
          call libQueueFuncs:push(qMoveBuffer,l_mTrajPt,l_bFlag)
        endIf
      endIf

      // process motion command from move buffer
      // @TODO move buffer should have elements previously interpolated to ensure they are 4 ms apart
      call libQueueFuncs:getNumElems(qMoveBuffer, l_nElems)
      if(l_nElems > 0)
        call libQueueFuncs:pop(qMoveBuffer,l_motion,l_bFlag)
        if(l_bFlag == true)
          nMovePts = nMovePts + 1

          // Velocity buffer to smooth out last traj point
          nVel[1] = nVel[0]
          nVel[0] = rosTrajPtMsg.jointTrajPt.nVelocity

          // Interpolate velocity for last point in trajectory
          call interpolateVel(l_motion)

          // contrary to what we did earlier, we unconditionally add the traj pt to the motion queue:
          // there doesn't appear to be a way to compare the 'current pose' of the robot to the pts
          // in the trajectory at the appropriate time (ie: when the robot is in motion and about to
          // start executing the segment towards 'l_motion').
          // Checking for dist(l_motion, herej()) (pseudo code) would not be correct as there will
          // always be a delay in the data coming out of herej() and the actual pose of the robot.
          // @TODO potentially set move id according to sequence value
          nMoveId = movej(l_motion.jJointRx, tTool, l_motion.mDesc)
        endIf
      endIf
    else
      // stop immediately -- resetMotion() also resets moveId
      resetMotion()
      // clear buffers
      call libQueueFuncs:clear(qTrajPtBuffer)
      call libQueueFuncs:clear(qMoveBuffer)
      bStopNow = false

      // debug
      nPtsPopped = 0
      nMovePts = 0
    endIf

    nMotionProgress = getMoveId()

    // sequence task
    delay(0)
  endWhile
end

--- motionCtrlVel.pgx ---
program motionCtrlVel()
  local bool l_bVelReady
  local num l_nIndex
  local num l_nResult
  local num l_nVelCmd[6]
begin
  // Copyright (c) 2021, Institute for Factory Automation and Production Systems (FAPS)
  //
  // Licensed under the Apache License, Version 2.0 (the "License");
  // you may not use this file except in compliance with the License.
  // You may obtain a copy of the License at
  //
  //     http://www.apache.org/licenses/LICENSE-2.0
  //
  // Unless required by applicable law or agreed to in writing, software
  // distributed under the License is distributed on an "AS IS" BASIS,
  // WITHOUT WARRANTIES OR CONDITIONS OF ANY KIND, either express or implied.
  // See the License for the specific language governing permissions and
  // limitations under the License.


  l_bVelReady=false

  while (true)
    // check connection status and whether to stop motion
    if (nConnFlagMotion==1 and nConnFlagState==1 and bStopNow==false)
      if (l_bVelReady==false)
		// start velocity mode according to configured velocity command type
        switch motionCfgVel.nCmdType
          case Staubli:VelocityType.JOINT
            $velJoint(motionCfgVel.tTool, motionCfgVel.mMaxSpeed)
            l_bVelReady=true
			if (bDebugMode and nDebugLevel==6)
				call printDebug("motionCtrlVel: $velJoint()",true)
			endIf
          break
          case Staubli:VelocityType.BASE_FRAME
            l_nResult=$velFrame(motionCfgVel.fReference, motionCfgVel.tTool, motionCfgVel.mMaxSpeed)
            if (l_nResult==0)
              l_bVelReady=true
            endIf
			if (bDebugMode and nDebugLevel==6)
				call printDebug("motionCtrlVel: $velFrame()",true)
				call printDebug("Result = "+toString("",l_nResult),false)
			endIf
          break
          case Staubli:VelocityType.TOOL_FRAME
            l_nResult=$velTool(motionCfgVel.tTool, motionCfgVel.mMaxSpeed)
            if (l_nResult==0)
              l_bVelReady=true
            endIf
            if (bDebugMode and nDebugLevel==6)
				call printDebug("motionCtrlVel: $velTool()",true)
				call printDebug("Result = "+toString("",l_nResult),false)
			endIf
          break
          default
            popUpMsg("Velocity motion command error: Unknown command type ("+toString("",motionCmdVel.nCmdType)+")")
          break
        endSwitch
      endIf

      if (l_bVelReady)
		// - copy global velocity command into local variable for $setVelCmd
		// - store velocity command in other global variable for UI
		// - reset global velocity command (fail-safe, avoiding repeated execution of old commands)
        for l_nIndex=0 to 5
          l_nVelCmd[l_nIndex]=motionCmdVel.nVelCmd[l_nIndex]
          actMotionCmdVel.nVelCmd[l_nIndex]=motionCmdVel.nVelCmd[l_nIndex]
          motionCmdVel.nVelCmd[l_nIndex]=0
        endFor

		// store velocity command type also for displaying in the UI
		actMotionCmdVel.nCmdType=motionCmdVel.nCmdType

        // execute velocity motion command
		$setVelCmd(l_nVelCmd)

        if (bDebugMode and nDebugLevel==6)
          call printDebug("motionCtrlVel: $setVelCmd()",true)
          call printDebug("l_nVelCmd = "+toString("",l_nVelCmd[0])+" "+toString("",l_nVelCmd[1])+" "+toString("",l_nVelCmd[2])+" "+toString("",l_nVelCmd[3])+" "+toString("",l_nVelCmd[4])+" "+toString("",l_nVelCmd[5])+" ",false)
        endIf
      endIf
    else
      // stop immediately -- resetMotion() also ends velocity mode
      resetMotion()
      l_bVelReady=false

      // set velocity motion command to initial state
      motionCmdVel.nSequence=0

      for l_nIndex=0 to 5
        motionCmdVel.nVelCmd[l_nIndex]=0
      endFor

      // debug
      if (bDebugMode and nDebugLevel==6)
        call printDebug("motionCtrlVel: resetMotion()",true)
        call printDebug("bStopNow: "+toString("",sel(bStopNow,1,0))+" inConn: "+toString("",nConnFlagMotion)+" outConn: "+toString("",nConnFlagState),false)
      endIf

      // reset stop flag
      bStopNow=false
    endIf

    // sequence task
    delay(0)
  endWhile
end

--- printDebug.pgx ---
public program printDebug(string x_sDebugMessage (dimensions=1), bool x_bStamp (dimensions=1))
begin
  // Copyright (c) 2021, Institute for Factory Automation and Production Systems (FAPS)
  //
  // Licensed under the Apache License, Version 2.0 (the "License");
  // you may not use this file except in compliance with the License.
  // You may obtain a copy of the License at
  //
  //     http://www.apache.org/licenses/LICENSE-2.0
  //
  // Unless required by applicable law or agreed to in writing, software
  // distributed under the License is distributed on an "AS IS" BASIS,
  // WITHOUT WARRANTIES OR CONDITIONS OF ANY KIND, either express or implied.
  // See the License for the specific language governing permissions and
  // limitations under the License.


  // check whether cursor is at last line (keys line)
  if (nDebugCursor==13)
    // erase line before printing the message
    put(scDebug,"                                        ")
    gotoxy(scDebug,0,13)
  endIf

  // print message
  if (x_bStamp)
    // print timestamp
    //put(scDebug,getDate("%H:%M:%S"))
    put(scDebug, "[" + toString(".3", clock()) + "] ")
  // else
    // put(scDebug,"  ")
  endIf
  putln(scDebug,x_sDebugMessage)
  nDebugCursor=sel(nDebugCursor==13,13,nDebugCursor+1)

  // update keys line if necessary
  if (nDebugCursor==13)
    gotoxy(scDebug,0,13)
    put(scDebug,"BACK")
    gotoxy(scDebug,16,13)
    put(scDebug,"CLS")
    gotoxy(scDebug,31,13)
    put(scDebug,"-")
    gotoxy(scDebug,36,13)
    put(scDebug,"+")
    gotoxy(scDebug,0,13)
  endIf
end

--- pushMotion.pgx ---
public program pushMotion(num& x_nMsgRecvState)
  local bool l_bOk
  local num l_nCounter
  local num l_nJointError
  local MotionCmd l_mTrajPt
begin
  // Copyright (c) 2016, Ocado Technology - Robotics Research Team
  //
  // Licensed under the Apache License, Version 2.0 (the "License");
  // you may not use this file except in compliance with the License.
  // You may obtain a copy of the License at
  //
  //     http://www.apache.org/licenses/LICENSE-2.0
  //
  // Unless required by applicable law or agreed to in writing, software
  // distributed under the License is distributed on an "AS IS" BASIS,
  // WITHOUT WARRANTIES OR CONDITIONS OF ANY KIND, either express or implied.
  // See the License for the specific language governing permissions and
  // limitations under the License.



  switch rosGenericMsg.header.nMsgType
    case nStdMsgType["JOINT_TRAJ_PT"]
      l_mTrajPt.nSequence=rosTrajPtMsg.jointTrajPt.nSeq

      // ROS joint position values are in rad, but VAL3 uses degrees
      call toJointRxDeg(rosTrajPtMsg.jointTrajPt.nJoints, l_mTrajPt.jJointRx)

      // from industrial_robot_client/src/joint_trajectory_interface.cpp
      // JointTrajectoryInterface::trajectory_to_msgs()
      // JointTrajectoryInterface::calc_speed()
      // velocity is converted to a scalar value representing % of max velocity,
      // such that 0.2 = 20% of maximum joint speed
      l_mTrajPt.mDesc.vel= limit((rosTrajPtMsg.jointTrajPt.nVelocity * 100), 0, 100)
      l_mTrajPt.nDuration=rosTrajPtMsg.jointTrajPt.nDuration

    break
    case nStdMsgType["JOINT_TRAJ_PT_FULL"]
      l_mTrajPt.nSequence=rosTrajPtFMsg.jointTrajPtFull.nSeq
      l_mTrajPt.nDuration=rosTrajPtFMsg.jointTrajPtFull.nTime

      // ROS joint position values are in rad, but VAL3 uses degrees
      call toJointRxDeg(rosTrajPtFMsg.jointTrajPtFull.nPositions, l_mTrajPt.jJointRx)

      // from industrial_robot_client/src/joint_trajectory_interface.cpp
      // JointTrajectoryInterface::trajectory_to_msgs()
      // JointTrajectoryInterface::calc_speed()
      // velocity is converted to a scalar value representing % of max velocity,
      // such that 0.2 = 20% of maximum joint speed
      l_mTrajPt.mDesc.vel= limit((rosTrajPtFMsg.jointTrajPtFull.nVelocities[0] * 100), 0, 100)
      // not sure about accelerations as yet
      l_mTrajPt.mDesc.accel=rosTrajPtFMsg.jointTrajPtFull.nAccelerations[0]
      l_mTrajPt.mDesc.decel=l_mTrajPt.mDesc.accel
    break
    default
    break
  endSwitch

  // see github.com/ros-industrial/industrial_core/simple_message/include/simple_message/joint_traj_pt.h
  if(l_mTrajPt.nSequence==-4)
    // set flag to stop immediately
    bStopNow=true
  else
    // check whether velocity value should be overwritten with value set on teach pendant
    if(bOverwriteVel == true)
      // overwrite velocity (and acceleration - ?)
      l_mTrajPt.mDesc.vel = getMonitorSpeed()
      // explicitly setting accel and decel to VAL3 default values
      l_mTrajPt.mDesc.accel = mNomSpeed.accel
      l_mTrajPt.mDesc.decel = mNomSpeed.decel
    endIf
    // only push motion into buffer if not a STOP message
    // and if joint positions are within software joint limits
    // and if velocity is greater than zero (beucase movej() will not accept vel <= 0)
    if(isInRange(l_mTrajPt.jJointRx) and l_mTrajPt.mDesc.vel > 0)
      call libQueueFuncs:push(qTrajPtBuffer,l_mTrajPt,l_bOk)
    else
      l_bOk = false
    endIf

    if(l_bOk==false)
      // could not push trajectory point into buffer
      // thus ACK should flag FAILURE, but only if comm type is request
      if(rosGenericMsg.header.nCommType==nCommType["SERVICE_REQUEST"])
        switch rosGenericMsg.header.nMsgType
          case nStdMsgType["JOINT_TRAJ_PT"]
            rosTrajPtAck.header.nReplyCode=2
          break
          case nStdMsgType["JOINT_TRAJ_PT_FULL"]
            rosTrajPtFAck.header.nReplyCode=2
          break
          default
          break
        endSwitch
      endIf
    endIf
  endIf
  // check whether ACK should be sent
  if(rosGenericMsg.header.nCommType == nCommType["SERVICE_REQUEST"])
    // comm type request requires ACK
    x_nMsgRecvState = nAck
  else
    // other comm types (e.g., topic) does not require ACK, hence skip state
    x_nMsgRecvState = nReset
  endIf
end

--- recvData.pgx ---
public program recvData(sio& x_sTcpSocket, num& x_nData[], num& x_nConnFlag, bool& x_bValidFlag)
  local num l_nByte
  local num l_nBytesRecv
  local num l_nIndex
begin
  // Copyright (c) 2016, Ocado Technology - Robotics Research Team
  // Copyright (c) 2021, Institute for Factory Automation and Production Systems (FAPS)
  //
  // Licensed under the Apache License, Version 2.0 (the "License");
  // you may not use this file except in compliance with the License.
  // You may obtain a copy of the License at
  //
  //     http://www.apache.org/licenses/LICENSE-2.0
  //
  // Unless required by applicable law or agreed to in writing, software
  // distributed under the License is distributed on an "AS IS" BASIS,
  // WITHOUT WARRANTIES OR CONDITIONS OF ANY KIND, either express or implied.
  // See the License for the specific language governing permissions and
  // limitations under the License.



  // attempt to receive data on specified socket

  // x_nConnFlag holds the current connection status of x_sTcpSocket

  l_nBytesRecv=0
  l_nIndex=0
  x_bValidFlag=false

  while (l_nBytesRecv<size(x_nData))
    l_nIndex=sioGet(x_sTcpSocket,l_nByte)
    if (l_nIndex==1)
      x_nData[l_nBytesRecv]=l_nByte
      l_nBytesRecv=l_nBytesRecv+1
      // received a byte, set flag to indicate connection
      x_nConnFlag=1
      // set global flag to indicate incoming data
      bDataIn=true
    elseIf (l_nIndex==-1)
      // error or timeout, indicate only if connection previously established
      if (x_nConnFlag==1)
        x_nConnFlag=-1
        // close connection properly (to avoid CLOSE_WAIT)
        clearBuffer(x_sTcpSocket)
      endIf
      return
    elseIf (l_nIndex == 0)
      // sioGet() returns 0 when connection is alive, thus set flag
      x_nConnFlag = 1
      if (l_nBytesRecv == 0)
        return
      endIf
    else
      // either < -1 or > 1
      popUpMsg("sioGet() returned " + toString("", l_nIndex))
      return
    endIf
  endWhile
  x_bValidFlag=true
end

--- recvHeartbeat.pgx ---
public program recvHeartbeat()
  local num l_nByte
  local num l_nBytesRecv
  local num l_nHtbt
  local num l_nHtbtB[4]
  local num l_nIndex
begin
  // Copyright (c) 2016, Ocado Technology - Robotics Research Team
  // Copyright (c) 2021, Institute for Factory Automation and Production Systems (FAPS)
  //
  // Licensed under the Apache License, Version 2.0 (the "License");
  // you may not use this file except in compliance with the License.
  // You may obtain a copy of the License at
  //
  //     http://www.apache.org/licenses/LICENSE-2.0
  //
  // Unless required by applicable law or agreed to in writing, software
  // distributed under the License is distributed on an "AS IS" BASIS,
  // WITHOUT WARRANTIES OR CONDITIONS OF ANY KIND, either express or implied.
  // See the License for the specific language governing permissions and
  // limitations under the License.



  while (true)
    l_nBytesRecv=0
    l_nIndex = sioGet(siTcpIpState, l_nByte)
    if (l_nIndex == -1)
      // connection not established or connection lost
      if (nConnFlagState == 1)
        nConnFlagState = -1
      endIf
    else
      // it means l_nIndex >= 0: connection established
      // check if connection had not already been established
      if (nConnFlagState != 1)
        // delay data output to avoid sync issues with client
        delay(1.0)
        // flag connection as established
        nConnFlagState = 1
      endIf
    endIf
  endWhile
end

--- recvMsgBody.pgx ---
public program recvMsgBody(sio& x_sSocket, num& x_nConnFlag, RosSimpleMsg& x_msg, num& x_nMsgRecvState)
  local bool l_bFlag
begin
  // Copyright (c) 2016, Ocado Technology - Robotics Research Team
  // Copyright (c) 2021, Institute for Factory Automation and Production Systems (FAPS)
  //
  // Licensed under the Apache License, Version 2.0 (the "License");
  // you may not use this file except in compliance with the License.
  // You may obtain a copy of the License at
  //
  //     http://www.apache.org/licenses/LICENSE-2.0
  //
  // Unless required by applicable law or agreed to in writing, software
  // distributed under the License is distributed on an "AS IS" BASIS,
  // WITHOUT WARRANTIES OR CONDITIONS OF ANY KIND, either express or implied.
  // See the License for the specific language governing permissions and
  // limitations under the License.



  l_bFlag=false

  switch x_msg.header.nMsgType
    // standard ROS industrial messages
    case SimpleMsg:MsgType.JOINT_TRAJ_PT
      call recvTrajPt(x_sSocket, x_nConnFlag, x_msg, l_bFlag)
    break
    case SimpleMsg:MsgType.JOINT_TRAJ_PT_F
      call recvTrajPtFull(x_sSocket,x_nConnFlag,x_msg,l_bFlag)
    break
    // Staubli specific
    case Staubli:MsgType.SET_DRIVE_POWER
      call recvRosMsg(x_sSocket, Staubli:setDrvPwrMsg.prefix, Staubli:setDrvPwrMsg.header, Staubli:setDrvPwrMsg.body, x_nConnFlag, x_msg, l_bFlag)
    break
    case Staubli:MsgType.WRITE_SINGLE_IO
      call recvRosMsg(x_sSocket, Staubli:writeSingIOMsg.prefix, Staubli:writeSingIOMsg.header, Staubli:writeSingIOMsg.body, x_nConnFlag, x_msg, l_bFlag)
    break
    case Staubli:MsgType.VELOCITY_CFG
      call recvRosMsg(x_sSocket, Staubli:velCfgMsg.prefix, Staubli:velCfgMsg.header, Staubli:velCfgMsg.body, x_nConnFlag, x_msg, l_bFlag)
    break
    case Staubli:MsgType.VELOCITY_CMD
      call recvRosMsg(x_sSocket, Staubli:velCmdMsg.prefix, Staubli:velCmdMsg.header, Staubli:velCmdMsg.body, x_nConnFlag, x_msg, l_bFlag)
    break
    default
      if (bDebugMode and nDebugLevel<=2)
        call printDebug("ERROR: unknown msg type ("+toString("",x_msg.header.nMsgType)+")",false)
      endIf
    break
  endSwitch

  if (l_bFlag == true)
    // move on to state 3: decode msg body
    x_nMsgRecvState = MsgRecvState.DECODE_BODY

    // debug
    if (bDebugMode and nDebugLevel<=2)
      call printDebug("INFO: receiving successful",false)
    endIf
  else
    // error whilst receiving msg body, reset state machine
    x_nMsgRecvState = MsgRecvState.RECEIVE_HEADER
    clearBuffer(x_sSocket)

    // debug
    if (bDebugMode and nDebugLevel<=2)
      call printDebug("ERROR: receiving not successful",false)
    endIf
  endIf
end

--- recvMsgHeader.pgx ---
public program recvMsgHeader(sio& x_sSocket (dimensions=1), num& x_nConnFlag (dimensions=1), RosSimpleMsg& x_msg (dimensions=1), num& x_nMsgRecvState (dimensions=1))
  local bool l_bFlag
begin
  // Copyright (c) 2016, Ocado Technology - Robotics Research Team
  // Copyright (c) 2021, Institute for Factory Automation and Production Systems (FAPS)
  //
  // Licensed under the Apache License, Version 2.0 (the "License");
  // you may not use this file except in compliance with the License.
  // You may obtain a copy of the License at
  //
  //     http://www.apache.org/licenses/LICENSE-2.0
  //
  // Unless required by applicable law or agreed to in writing, software
  // distributed under the License is distributed on an "AS IS" BASIS,
  // WITHOUT WARRANTIES OR CONDITIONS OF ANY KIND, either express or implied.
  // See the License for the specific language governing permissions and
  // limitations under the License.



  // attempt to receive message prefix and header
  call recvData(x_sSocket,x_msg.prefix.nData,x_nConnFlag,l_bFlag)
  if (l_bFlag==true)
    call recvData(x_sSocket,x_msg.header.nData,x_nConnFlag,l_bFlag)
  endIf

  if (l_bFlag == true)
    // move on to state 1: decode header
    x_nMsgRecvState = MsgRecvState.DECODE_HEADER
  else
    // error: reset state to 0: receive header
    x_nMsgRecvState = MsgRecvState.RECEIVE_HEADER
  endIf
end

--- recvRosMsg.pgx ---
program recvRosMsg(sio& x_sSocket (dimensions=1), Prefix& x_pPrefix (dimensions=1), Header& x_hHeader (dimensions=1), Body& x_bBody (dimensions=1), num& x_nConnFlag (dimensions=1), RosSimpleMsg& x_msg (dimensions=1), bool& x_bValidFlag (dimensions=1))
begin
  // Copyright (c) 2021, Institute for Factory Automation and Production Systems (FAPS)
  //
  // Licensed under the Apache License, Version 2.0 (the "License");
  // you may not use this file except in compliance with the License.
  // You may obtain a copy of the License at
  //
  //     http://www.apache.org/licenses/LICENSE-2.0
  //
  // Unless required by applicable law or agreed to in writing, software
  // distributed under the License is distributed on an "AS IS" BASIS,
  // WITHOUT WARRANTIES OR CONDITIONS OF ANY KIND, either express or implied.
  // See the License for the specific language governing permissions and
  // limitations under the License.


  // attempt to receive the data of the message (prefix and header are in x_msg)
  x_pPrefix.nLength=x_msg.prefix.nLength
  x_hHeader.nMsgType=x_msg.header.nMsgType
  x_hHeader.nCommType=x_msg.header.nCommType
  x_hHeader.nReplyCode=x_msg.header.nReplyCode

  call recvData(x_sSocket,x_bBody.nData,x_nConnFlag,x_bValidFlag)
end

--- recvTrajPt.pgx ---
public program recvTrajPt(sio& x_sSocket (dimensions=1), num& x_nConnFlag (dimensions=1), RosSimpleMsg& x_msg (dimensions=1), bool& x_bFlag (dimensions=1))
begin
  // Copyright (c) 2016, Ocado Technology - Robotics Research Team
  // Copyright (c) 2021, Institute for Factory Automation and Production Systems (FAPS)
  //
  // Licensed under the Apache License, Version 2.0 (the "License");
  // you may not use this file except in compliance with the License.
  // You may obtain a copy of the License at
  //
  //     http://www.apache.org/licenses/LICENSE-2.0
  //
  // Unless required by applicable law or agreed to in writing, software
  // distributed under the License is distributed on an "AS IS" BASIS,
  // WITHOUT WARRANTIES OR CONDITIONS OF ANY KIND, either express or implied.
  // See the License for the specific language governing permissions and
  // limitations under the License.



  // attempt to receive message ID 11 data (prefix and header are in x_msg)
  rosTrajPtMsg.prefix.nLength=x_msg.prefix.nLength
  rosTrajPtMsg.header.nMsgType=x_msg.header.nMsgType
  rosTrajPtMsg.header.nCommType=x_msg.header.nCommType
  rosTrajPtMsg.header.nReplyCode=x_msg.header.nReplyCode

  call recvData(x_sSocket,rosTrajPtMsg.body.nData,x_nConnFlag,x_bFlag)
end

--- recvTrajPtFull.pgx ---
public program recvTrajPtFull(sio& x_sSocket (dimensions=1), num& x_nConnFlag (dimensions=1), RosSimpleMsg& x_msg (dimensions=1), bool& x_bFlag (dimensions=1))
begin
  // Copyright (c) 2016, Ocado Technology - Robotics Research Team
  // Copyright (c) 2021, Institute for Factory Automation and Production Systems (FAPS)
  //
  // Licensed under the Apache License, Version 2.0 (the "License");
  // you may not use this file except in compliance with the License.
  // You may obtain a copy of the License at
  //
  //     http://www.apache.org/licenses/LICENSE-2.0
  //
  // Unless required by applicable law or agreed to in writing, software
  // distributed under the License is distributed on an "AS IS" BASIS,
  // WITHOUT WARRANTIES OR CONDITIONS OF ANY KIND, either express or implied.
  // See the License for the specific language governing permissions and
  // limitations under the License.



  // receive message ID 14 data (prefix and header are in x_msg)
  rosTrajPtFMsg.prefix.nLength=x_msg.prefix.nLength
  rosTrajPtFMsg.header.nMsgType=x_msg.header.nMsgType
  rosTrajPtFMsg.header.nCommType=x_msg.header.nCommType
  rosTrajPtFMsg.header.nReplyCode=x_msg.header.nReplyCode

  call recvData(x_sSocket,rosTrajPtFMsg.body.nData,x_nConnFlag,x_bFlag)
end

--- screenUpdate.pgx ---
public program screenUpdate(num x_nPeriod (dimensions=1))
  local num l_nElems
  local num l_nExecStatus
  local num l_nKey
  local num l_nIdx
  local string l_sVelCmdType
begin
  // Copyright (c) 2016, Ocado Technology - Robotics Research Team
  // Copyright (c) 2021, Institute for Factory Automation and Production Systems (FAPS)
  //
  // Licensed under the Apache License, Version 2.0 (the "License");
  // you may not use this file except in compliance with the License.
  // You may obtain a copy of the License at
  //
  //     http://www.apache.org/licenses/LICENSE-2.0
  //
  // Unless required by applicable law or agreed to in writing, software
  // distributed under the License is distributed on an "AS IS" BASIS,
  // WITHOUT WARRANTIES OR CONDITIONS OF ANY KIND, either express or implied.
  // See the License for the specific language governing permissions and
  // limitations under the License.


  // screen status indicator
  l_nExecStatus=0

  // setup debug screen
  nDebugLevel=5
  nDebugLevelMax=8
  bDebugMode=false
  cls(scDebug)
  title(scDebug,"ROS-I server (DEBUG: Level "+toString("",nDebugLevel)+")")
  gotoxy(scDebug,0,13)
  put(scDebug,"BACK")
  gotoxy(scDebug,16,13)
  put(scDebug,"CLS")
  gotoxy(scDebug,31,13)
  put(scDebug,"-")
  gotoxy(scDebug,36,13)
  put(scDebug,"+")
  gotoxy(scDebug,0,0)
  nDebugCursor=0

  // setup main screen
  userPage(scMonitor)
  cls(scMonitor)
  title(scMonitor,"ROS-I server")

  while (true)
    // check whether debug screen is enabled
    if (bDebugMode)
      // -----------------------------------------------------
      // DEBUG SCREEN
      // -----------------------------------------------------
      // show the debug screen if not done already
      if (!bShowDebug)
        userPage(scDebug)
        bShowDebug=true
      endIf

      l_nKey=getKey(scDebug)

      switch (l_nKey)
        // toggle screen with F1
        case 271
          bShowDebug=false
          bDebugMode=false
          userPage(scMonitor)
        break
        // clear debug screen with F4
        case 274
          cls(scDebug)
          gotoxy(scDebug,0,13)
          put(scDebug,"BACK")
          gotoxy(scDebug,16,13)
          put(scDebug,"CLS")
          gotoxy(scDebug,31,13)
          put(scDebug,"-")
          gotoxy(scDebug,36,13)
          put(scDebug,"+")
          gotoxy(scDebug,0,0)
          nDebugCursor=0
        break
        // decrease debug level with F7
        case 277
          nDebugLevel=sel(nDebugLevel==0,0,nDebugLevel-1)
          title(scDebug,"ROS-I server (DEBUG: Level "+toString("",nDebugLevel)+")")
        break
        // increase debug level with F8
        case 278
          nDebugLevel=sel(nDebugLevel==nDebugLevelMax,nDebugLevelMax,nDebugLevel+1)
          title(scDebug,"ROS-I server (DEBUG: Level "+toString("",nDebugLevel)+")")
        break
        // ignore other keys
        default
        break
      endSwitch

    else
      // -----------------------------------------------------
      // MAIN SCREEN
      // -----------------------------------------------------
      // clear screen and set title
      cls(scMonitor)
      switch (nMotionMode)
        case Staubli:MotionMode.JOINT_TRAJ
          title(scMonitor,"ROS-I server [JOINT_TRAJECTORY]")
        break
        case Staubli:MotionMode.VELOCITY_CTRL
          title(scMonitor,"ROS-I server [VELOCITY_CONTROL]")
        break
        default
          title(scMonitor,"ROS-I server")
        break
      endSwitch

      // toggle velocity overwrite upon release of F7/F8 keys
      l_nKey=getKey(scMonitor)
      call libQueueFuncs:getNumElems(qMoveBuffer,l_nElems)
      if (l_nKey==277 and bOverwriteVel==false)
        if (l_nElems==0)
          bOverwriteVel=true
        else
          popUpMsg("Motion buffer not empty; cannot enable V/OW")
        endIf
      elseIf (l_nKey==278 and bOverwriteVel==true)
        if (l_nElems==0)
          bOverwriteVel=false
        else
          popUpMsg("Motion buffer not empty; cannot disable V/OW")
        endIf
      endIf

      // switch to debug screen upon release of F1 key
      if (l_nKey==271)
        bDebugMode=true
      endIf

      // update connection status on port 11000
      gotoxy(scMonitor,0,0)
      // 15 characters: gotoxy(16,0) to insert status
      put(scMonitor,"Motion (11000):")
      gotoxy(scMonitor,16,0)
      switch nConnFlagMotion
        case -1
          put(scMonitor,"connection lost")
        break
        case 0
          put(scMonitor,"not connected")
        break
        case 1
          put(scMonitor,"connected")
        break
        default
          put(scMonitor,"not connected")
        break
      endSwitch
      // update data incoming indicator
      if (bDataIn)
        gotoxy(scMonitor,37,0)
        put(scMonitor,"<<<")
        bDataIn=false
      endIf

      // update connection status on port 11001
      gotoxy(scMonitor,0,1)
      // 15 characters: gotoxy(16,0) to insert status
      put(scMonitor,"System (11001):")
      gotoxy(scMonitor,16,1)
      switch nConnFlagSystem
        case -1
          put(scMonitor,"connection lost")
        break
        case 0
          put(scMonitor,"not connected")
        break
        case 1
          put(scMonitor,"connected")
        break
        default
          put(scMonitor,"not connected")
        break
      endSwitch

      // update connection status on port 11002
      gotoxy(scMonitor,0,2)
      // 15 characters: gotoxy(16,2) to insert status
      put(scMonitor,"State  (11002):")
      gotoxy(scMonitor,16,2)
      switch nConnFlagState
        case -1
          put(scMonitor,"connection lost")
        break
        case 0
          put(scMonitor,"not connected")
        break
        case 1
          put(scMonitor,"connected")
        break
        default
          put(scMonitor,"not connected")
        break
      endSwitch
      // update data outgoing indicator
      if (bDataOut)
        gotoxy(scMonitor,37,2)
        put(scMonitor,">>>")
        bDataOut=false
      endIf

      // update connection status on port 11003
      gotoxy(scMonitor,0,3)
      // 15 characters: gotoxy(16,3) to insert status
      put(scMonitor,"IO     (11003):")
      gotoxy(scMonitor,16,3)
      switch nConnFlagIO
        case -1
          put(scMonitor,"connection lost")
        break
        case 0
          put(scMonitor,"not connected")
        break
        case 1
          put(scMonitor,"connected")
        break
        default
          put(scMonitor,"not connected")
        break
      endSwitch

      if (nMotionMode == Staubli:MotionMode.JOINT_TRAJ)
        // update trajectory buffer size
        call libQueueFuncs:getNumElems(qTrajPtBuffer,l_nElems)
        gotoxy(scMonitor,0,5)
        // 18 characteres: gotoxy(19,3) to insert status
        put(scMonitor,"Trajectory buffer:")
        gotoxy(scMonitor,19,5)
        put(scMonitor,l_nElems)
        // also print number of points popped from buffer
        gotoxy(scMonitor,24,5)
        put(scMonitor,nPtsPopped)
        // do the same for move buffer
        call libQueueFuncs:getNumElems(qMoveBuffer,l_nElems)
        gotoxy(scMonitor,0,6)
        put(scMonitor,"Motion buffer:")
        gotoxy(scMonitor,19,6)
        put(scMonitor,l_nElems)
        gotoxy(scMonitor,24,6)
        put(scMonitor,nMovePts)

        // display velocity overwrite status
        gotoxy(scMonitor,0,7)
        put(scMonitor,"Velocity overwrite:")
        gotoxy(scMonitor,20,7)
        if (bOverwriteVel==true)
          put(scMonitor,"enabled")
        else
          put(scMonitor,"disabled")
        endIf

        // display nMoveId and nMotionProgress
        gotoxy(scMonitor,0,8)
        put(scMonitor,"moveId:")
        gotoxy(scMonitor,8,8)
        put(scMonitor,nMoveId)
        gotoxy(scMonitor,13,8)
        put(scMonitor,"progress:")
        gotoxy(scMonitor,23,8)
        put(scMonitor,nMotionProgress)

      elseIf (nMotionMode == Staubli:MotionMode.VELOCITY_CTRL)
        // get velocity command type as string
        switch actMotionCmdVel.nCmdType
          case Staubli:VelocityType.INVALID
            l_sVelCmdType = "INVALID"
          break
          case Staubli:VelocityType.JOINT
            l_sVelCmdType = "JOINT"
          break
          case Staubli:VelocityType.BASE_FRAME
            l_sVelCmdType = "BASE_FRAME"
          break
          case Staubli:VelocityType.TOOL_FRAME
            l_sVelCmdType = "TOOL_FRAME"
          break
          default
            l_sVelCmdType = "Unknown=" + toString("", actMotionCmdVel.nCmdType)
          break
        endSwitch
        // print velocity command data and type
        gotoxy(scMonitor, 0, 5)
        put(scMonitor, "Velocity Command (" + l_sVelCmdType + "):")
        for l_nIdx = 0 to 5
          gotoxy(scMonitor, l_nIdx * 7, 6)
          put(scMonitor, toString("5", actMotionCmdVel.nVelCmd[l_nIdx]))
        endFor
        // print velocity config data
        gotoxy(scMonitor, 0, 7)
        put(scMonitor, "Velocity Config (accel,vel,tvel,rvel):")
        gotoxy(scMonitor, 0, 8)
        put(scMonitor, "a: "+toString("",motionCfgVel.mMaxSpeed.accel)+" | v: "+toString("",motionCfgVel.mMaxSpeed.vel)+" | t: "+toString("",motionCfgVel.mMaxSpeed.tvel)+" | r: "+toString("",motionCfgVel.mMaxSpeed.rvel))
      endIf



      // display time between valid trajectory point received and ACK sent
      gotoxy(scMonitor,0,10)
      put(scMonitor,"recvMsgHeader:")
      gotoxy(scMonitor,15,10)
      put(scMonitor,toString(".3",nHeaderTime))

      gotoxy(scMonitor,0,11)
      put(scMonitor,"other states:")
      gotoxy(scMonitor,15,11)
      put(scMonitor,toString(".4",nElapsedTime))

      // update debug status
      gotoxy(scMonitor,37,11)
      switch l_nExecStatus
        case 0
          put(scMonitor,"[+]")
          l_nExecStatus=1
        break
        case 1
          put(scMonitor,"[-]")
          l_nExecStatus=0
        break
        default
        break
      endSwitch

      // add Function keys labels
      gotoxy(scMonitor,0,13)
      put(scMonitor,"DBG")
      gotoxy(scMonitor,30,13)
      put(scMonitor,"V/ON")
      gotoxy(scMonitor,35,13)
      put(scMonitor,"V/OFF")

    endIf

    // sequence task
    delay(x_nPeriod)
  endWhile
end

--- sendAck.pgx ---
public program sendAck(sio& x_sSocket, num& x_nConnFlag, RosSimpleMsg& x_msg, num& x_nMsgRecvState)
begin
  // Copyright (c) 2016, Ocado Technology - Robotics Research Team
  // Copyright (c) 2021, Institute for Factory Automation and Production Systems (FAPS)
  //
  // Licensed under the Apache License, Version 2.0 (the "License");
  // you may not use this file except in compliance with the License.
  // You may obtain a copy of the License at
  //
  //     http://www.apache.org/licenses/LICENSE-2.0
  //
  // Unless required by applicable law or agreed to in writing, software
  // distributed under the License is distributed on an "AS IS" BASIS,
  // WITHOUT WARRANTIES OR CONDITIONS OF ANY KIND, either express or implied.
  // See the License for the specific language governing permissions and
  // limitations under the License.



  switch x_msg.header.nMsgType
    case SimpleMsg:MsgType.JOINT_TRAJ_PT
      call sendRosMsg(x_sSocket, rosTrajPtAck.prefix, rosTrajPtAck.header, rosTrajPtAck.body, x_nConnFlag)
    break
    case SimpleMsg:MsgType.JOINT_TRAJ_PT_F
      call sendRosMsg(x_sSocket, rosTrajPtFAck.prefix, rosTrajPtFAck.header, rosTrajPtFAck.body, x_nConnFlag)
    break
    // Staubli specific
    case Staubli:MsgType.SET_DRIVE_POWER
      call sendRosMsg(x_sSocket, Staubli:setDrvPwrAck.prefix, Staubli:setDrvPwrAck.header, Staubli:setDrvPwrAck.body, x_nConnFlag)
    break
    case Staubli:MsgType.WRITE_SINGLE_IO
      call sendRosMsg(x_sSocket, Staubli:writeSingIOAck.prefix, Staubli:writeSingIOAck.header, Staubli:writeSingIOAck.body, x_nConnFlag)
    break
    case Staubli:MsgType.VELOCITY_CFG
      call sendRosMsg(x_sSocket, Staubli:velCfgAck.prefix, Staubli:velCfgAck.header, Staubli:velCfgAck.body, x_nConnFlag)
    break
    case Staubli:MsgType.VELOCITY_CMD
      call sendRosMsg(x_sSocket, Staubli:velCmdAck.prefix, Staubli:velCmdAck.header, Staubli:velCmdAck.body, x_nConnFlag)
    break
    // default
    default
      //region @DEBUG
      if (bDebugMode and nDebugLevel<=5)
        call printDebug("sendAck: switch (msgType)",true)
        call printDebug("ERROR: unknown msg type",false)
      endIf
      //endregion
    break
  endSwitch

  // regardless of result from sending ACK
  // reset state machine to receive new messages
  x_nMsgRecvState = MsgRecvState.RECEIVE_HEADER
end

--- sendData.pgx ---
public program sendData(sio& x_sTcpSocket, num& x_nData[], num& x_nFlag)
  local num l_nRetVal
begin
  // Copyright (c) 2016, Ocado Technology - Robotics Research Team
  // Copyright (c) 2021, Institute for Factory Automation and Production Systems (FAPS)
  //
  // Licensed under the Apache License, Version 2.0 (the "License");
  // you may not use this file except in compliance with the License.
  // You may obtain a copy of the License at
  //
  //     http://www.apache.org/licenses/LICENSE-2.0
  //
  // Unless required by applicable law or agreed to in writing, software
  // distributed under the License is distributed on an "AS IS" BASIS,
  // WITHOUT WARRANTIES OR CONDITIONS OF ANY KIND, either express or implied.
  // See the License for the specific language governing permissions and
  // limitations under the License.



  // send data via socket connection...
  // but only if connection is alive
  if (x_nFlag == 1)
    l_nRetVal=sioSet(x_sTcpSocket,x_nData)
    if (l_nRetVal==-1)
      if (x_nFlag==1)
        x_nFlag=-1
      endIf
    elseIf (l_nRetVal<size(x_nData))
      popUpMsg("Error while sending data")
      x_nFlag=-1
    else
      bDataOut=true
    endIf
  endIf
end

--- stateMachine.pgx ---
program stateMachine()
  local bool l_bKillMotTask
  local bool l_bOk
  local bool l_bResetMotion
  local num l_nNextState
begin
  // Copyright (c) 2021, Institute for Factory Automation and Production Systems (FAPS)
  //
  // Licensed under the Apache License, Version 2.0 (the "License");
  // you may not use this file except in compliance with the License.
  // You may obtain a copy of the License at
  //
  //     http://www.apache.org/licenses/LICENSE-2.0
  //
  // Unless required by applicable law or agreed to in writing, software
  // distributed under the License is distributed on an "AS IS" BASIS,
  // WITHOUT WARRANTIES OR CONDITIONS OF ANY KIND, either express or implied.
  // See the License for the specific language governing permissions and
  // limitations under the License.


  while (true)
    // assume success to state transition
    l_bOk=true
    // reset flags
    l_bKillMotTask=false
    l_bResetMotion=false
    // wait for state transition event
    wait(bMotionMsgEvent)
    bMotionMsgEvent=false

    // //region @DEBUG
    // if (bDebugMode and nDebugLevel==7)
      // call printDebug("stateMachine: got event ("+toString("",nMotionMsgType)+")",true)
      // call printDebug("INFO: current state: "+toString("",nMotionMode),false)
    // endIf
    // //endregion

    //region @switch_current_state -- check whether the current motion task has to be killed
    //                                and set next state
    if (nMotionMode==Staubli:MotionMode.JOINT_TRAJ)

      switch (nMotionMsgType)
        case SimpleMsg:MsgType.JOINT_TRAJ_PT,SimpleMsg:MsgType.JOINT_TRAJ_PT_F
          // already in JOINT_TRAJ mode, skip state transition
          l_bOk=false
        break
        case Staubli:MsgType.VELOCITY_CFG
          l_bKillMotTask=true
          l_nNextState=Staubli:MotionMode.VELOCITY_CTRL
        break
      endSwitch

    elseIf (nMotionMode==Staubli:MotionMode.VELOCITY_CTRL)

      switch (nMotionMsgType)
        case SimpleMsg:MsgType.JOINT_TRAJ_PT,SimpleMsg:MsgType.JOINT_TRAJ_PT_F
          l_bKillMotTask=true
          l_nNextState=Staubli:MotionMode.JOINT_TRAJ
        break
        case Staubli:MsgType.VELOCITY_CFG
          l_bResetMotion=true
        break
      endSwitch

    endIf
    //endregion @switch_current_state

